// TIA Portal V15 export
// export: Created 2018-05-30T14:06:48.0973328Z, ExportSetting WithDefaults, WithReadOnly, DisplayName Totally Integrated Automation Portal, DisplayVersion V15, DisplayName STEP 7 Professional, DisplayVersion V15, DisplayName WinCC Professional, DisplayVersion V15, DisplayName TIA Portal Openness, DisplayVersion V15
FUNCTION_BLOCK "BST_DIGITAL_400"   // FB24, STL
{ S7_Optimized_Access := 'FALSE' }
VERSION : 0.1
// stored: AutoNumber false, CodeModifiedDate 2018-05-30T14:06:41.0879319Z, CompileDate 2018-05-30T14:06:41.0879318Z, CreationDate 2018-05-30T13:57:30.9234642Z, InterfaceModifiedDate 2018-05-30T14:02:05.4231647Z, IsConsistent true, IsKnowHowProtected false, ISMultiInstanceCapable true, IsWriteProtected false, LibraryConformanceStatus The object is library-conformant., ModifiedDate 2018-05-30T14:06:41.0879319Z, ParameterModified 2018-05-30T14:02:05.4231647Z, StructureModified 2018-05-30T14:02:05.4231647Z, UDAEnableTagReadback false
   VAR_INPUT
      i_bInp : Bool;
   END_VAR
   VAR_OUTPUT
      QON : Bool;
   END_VAR
BEGIN
END_FUNCTION_BLOCK
